// TIA Portal project "一个开关控制两个灯" (V16)

(* hardware
DEVICE "S7-1200 station_1"  S7-1200 Station
   slot 0: "Rack_0"  S7-1200 Rack  Rack  V1.0
   slot 1: "PLC_1"  CPU 1214C DC/DC/DC  6ES7 214-1AG40-0XB0  V4.4
DEVICE "HMI_1"  KTP700 Basic PN
   slot 0: "HMI_1"  KTP700 Basic PN  6AV2 123-2GB03-0AX0  16.0.0.0
   slot 1: "HMI_RT_1"  KTP700 Basic PN  6AV2 123-2GB03-0AX0  16.0.0.0
   slot 5: "HMI_1.IE_CP_1"  PROFINET Interface  16.0.0.0
      slot 1: "PROFINET Interface_1"  PROFINET Interface
         slot 1: "Port_1"  Port
*)

// ===== PLC "PLC_1"  CPU 1214C DC/DC/DC =====

VAR_GLOBAL   // PLC tag table "默认变量表"
   "Tag_1" AT %M0.0 : Bool;
   "Tag_2" AT %M0.1 : Bool;
   "Tag_3" AT %M0.2 : Bool;
   "Tag_4" AT %Q0.1 : Bool;
   "Tag_5" AT %Q0.2 : Bool;
   "Tag_6" AT %M10.0 : Bool;
   "Tag_7" AT %M10.1 : Bool;
   "Tag_8" AT %Q0.7 : Bool;
   "Tag_9" AT %M1.0 : Bool;
   "Tag_10" AT %M1.1 : Bool;
   "Tag_11" AT %M1.2 : Bool;
   "Tag_12" AT %M1.3 : Bool;
   "Tag_13" AT %M1.4 : Bool;
   "Tag_14" AT %Q0.0 : Bool;
   "Tag_15" AT %M2.0 : Bool;
   "Tag_16" AT %M2.1 : Bool;
   "Tag_17" AT %M2.2 : Bool;
   "Tag_18" AT %I0.0 : Bool;
   "Tag_19" AT %Q1.0 : Bool;
   "Tag_20" AT %Q1.1 : Bool;
   "Tag_21" AT %M1.5 : Bool;
   "Tag_22" AT %M1.6 : Bool;
   "Tag_23" AT %M1.7 : Bool;
END_VAR

DATA_BLOCK "数据块_1"   // DB2
{ S7_Optimized_Access := 'TRUE' }
VERSION : 0.1
   VAR
      中间变量1 : Bool;
      中间变量2 : Bool;
      中间变量3 : Bool;
      中间变量4 : Bool;
      中间变量5 : Bool;
      中间变量6 : Bool;
      中间变量7 : Bool;
      中间变量8 : Bool;
      数值 : UDInt := 2;
      上升 : Array[1..10] of Bool;
      下降 : Array[1..10] of Bool;
      中间1 : Array[1..10] of Bool;
   END_VAR
BEGIN
END_DATA_BLOCK

// folder: System blocks/Program resources

DATA_BLOCK "IEC_Counter_0_DB"   // DB1
{ S7_Optimized_Access := 'TRUE' }
AUTHOR : Simatic
FAMILY : IEC
NAME : CNTR
VERSION : 1.0
// stored: InstanceOfName IEC_COUNTER
"IEC_COUNTER"
BEGIN
END_DATA_BLOCK

DATA_BLOCK "IEC_Counter_0_DB_1"   // DB3
{ S7_Optimized_Access := 'TRUE' }
AUTHOR : Simatic
FAMILY : IEC
NAME : CNTR
VERSION : 1.0
// stored: InstanceOfName IEC_COUNTER
"IEC_COUNTER"
BEGIN
END_DATA_BLOCK

DATA_BLOCK "IEC_Counter_0_DB_2"   // DB4
{ S7_Optimized_Access := 'TRUE' }
AUTHOR : Simatic
FAMILY : IEC
NAME : CNTR
VERSION : 1.0
// stored: InstanceOfName IEC_COUNTER
"IEC_COUNTER"
BEGIN
END_DATA_BLOCK

// folder: (top level)

FUNCTION "MHJ-PLC-Lab-Function-S71200" : Void   // FC9000, SCL
{ S7_Optimized_Access := 'TRUE' }
VERSION : 0.1
   VAR_TEMP
      rdTimeReturn : Int;
      outputTime : DTL;
      SyncVal : Byte;
      forVal : Int;
      forVal_2 : Int;
      Value : Byte;
   END_VAR
   VAR CONSTANT
      CompVal : Byte := 16#34;
      Value_01 : Byte := 16#11;
      Value_01_DW : DWord := 16#A165_D992;
      Value_02_DW : DWord := 16#58BE_4401;
   END_VAR
BEGIN

   #Value:=PEEK(area := 16#82,
        dbNumber := 0,
        byteOffset := 511);
   #Value := #Value + 1;

   POKE(area := 16#82,
        dbNumber := 0,
        byteOffset := 511,
        value := #Value);

   POKE(area:=16#81,
        dbNumber:=0,
        byteOffset:=1016,
        value:=#Value_01_DW);
   POKE(area := 16#81,
        dbNumber := 0,
        byteOffset := 1020,
        value := #Value_02_DW);

   POKE(area := 16#81,
        dbNumber := 0,
        byteOffset := 511,
        value := B#16#00);

   FOR #forVal := 0 TO 120 DO
       FOR #forVal_2:=0 TO 10 DO
           #rdTimeReturn:=RD_SYS_T(#outputTime);
           #rdTimeReturn := WR_SYS_T(#outputTime);
           #rdTimeReturn := RD_SYS_T(#outputTime);
           #rdTimeReturn := WR_SYS_T(#outputTime);
       END_FOR;
       #SyncVal:= PEEK(area := 16#81,
                      dbNumber := 0,
                      byteOffset := 511);
       IF #SyncVal = #CompVal THEN
          GOTO M_1;
       END_IF;
   END_FOR;
   RETURN;

   M_1:
   POKE(area := 16#81,
        dbNumber := 0,
        byteOffset := 511,
        value := B#16#0);
END_FUNCTION

ORGANIZATION_BLOCK "Main"   // OB1, LAD, ProgramCycle
TITLE = "Main Program Sweep (Cycle)"
{ S7_Optimized_Access := 'TRUE' }
VERSION : 0.1
   VAR_INPUT
      Initial_Call : Bool;   // Initial call of this OB
      Remanence : Bool;   // =True, if remanent data are available
   END_VAR
   VAR_TEMP   // added for the SCL form of the ladder/FBD networks
      _w1 : Bool;
      _w2 : Bool;
      _w3 : Bool;
      _w4 : Bool;
   END_VAR
BEGIN

REGION Network 1
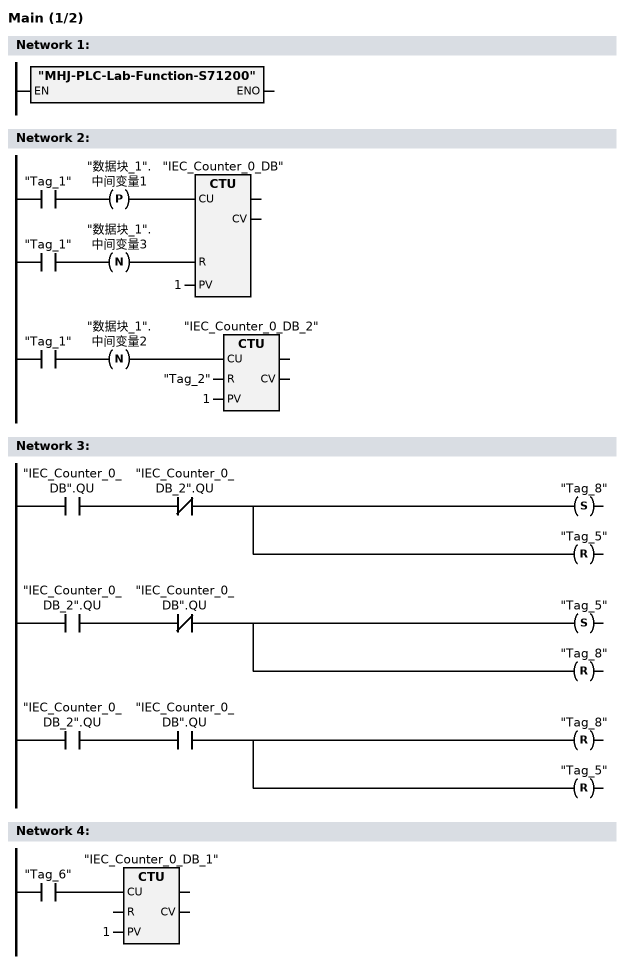
   RUNG wire#powerrail
      "MHJ-PLC-Lab-Function-S71200"()
   END_RUNG
   // the same network as SCL:
   "MHJ-PLC-Lab-Function-S71200"();
END_REGION

REGION Network 2
   #_w1 := "Tag_1" AND NOT "数据块_1".中间变量1;   // rising edge
   "数据块_1".中间变量1 := "Tag_1";
   #_w2 := NOT "Tag_1" AND "数据块_1".中间变量3;   // falling edge
   "数据块_1".中间变量3 := "Tag_1";
   "IEC_Counter_0_DB".CTU(CU := #_w1, R := #_w2, PV := 1);
   #_w3 := NOT "Tag_1" AND "数据块_1".中间变量2;   // falling edge
   "数据块_1".中间变量2 := "Tag_1";
   "IEC_Counter_0_DB_2".CTU(CU := #_w3, R := "Tag_2", PV := 1);
END_REGION

REGION Network 3
   RUNG wire#powerrail
      Contact( "IEC_Counter_0_DB".QU )
      I_Contact( "IEC_Counter_0_DB_2".QU )
      wire#w1
      S_Coil( "Tag_8" )
   END_RUNG
   RUNG wire#w1
      R_Coil( "Tag_5" )
   END_RUNG
   RUNG wire#powerrail
      Contact( "IEC_Counter_0_DB_2".QU )
      I_Contact( "IEC_Counter_0_DB".QU )
      wire#w2
      S_Coil( "Tag_5" )
   END_RUNG
   RUNG wire#w2
      R_Coil( "Tag_8" )
   END_RUNG
   RUNG wire#powerrail
      Contact( "IEC_Counter_0_DB_2".QU )
      Contact( "IEC_Counter_0_DB".QU )
      wire#w3
      R_Coil( "Tag_8" )
   END_RUNG
   RUNG wire#w3
      R_Coil( "Tag_5" )
   END_RUNG
   // the same network as SCL:
   IF "IEC_Counter_0_DB".QU AND NOT "IEC_Counter_0_DB_2".QU THEN
       "Tag_8" := TRUE;
       "Tag_5" := FALSE;
   END_IF;
   IF "IEC_Counter_0_DB_2".QU AND NOT "IEC_Counter_0_DB".QU THEN
       "Tag_5" := TRUE;
       "Tag_8" := FALSE;
   END_IF;
   IF "IEC_Counter_0_DB_2".QU AND "IEC_Counter_0_DB".QU THEN
       "Tag_8" := FALSE;
       "Tag_5" := FALSE;
   END_IF;
END_REGION

REGION Network 4
   "IEC_Counter_0_DB_1".CTU(CU := "Tag_6", PV := 1);
END_REGION

REGION Network 5
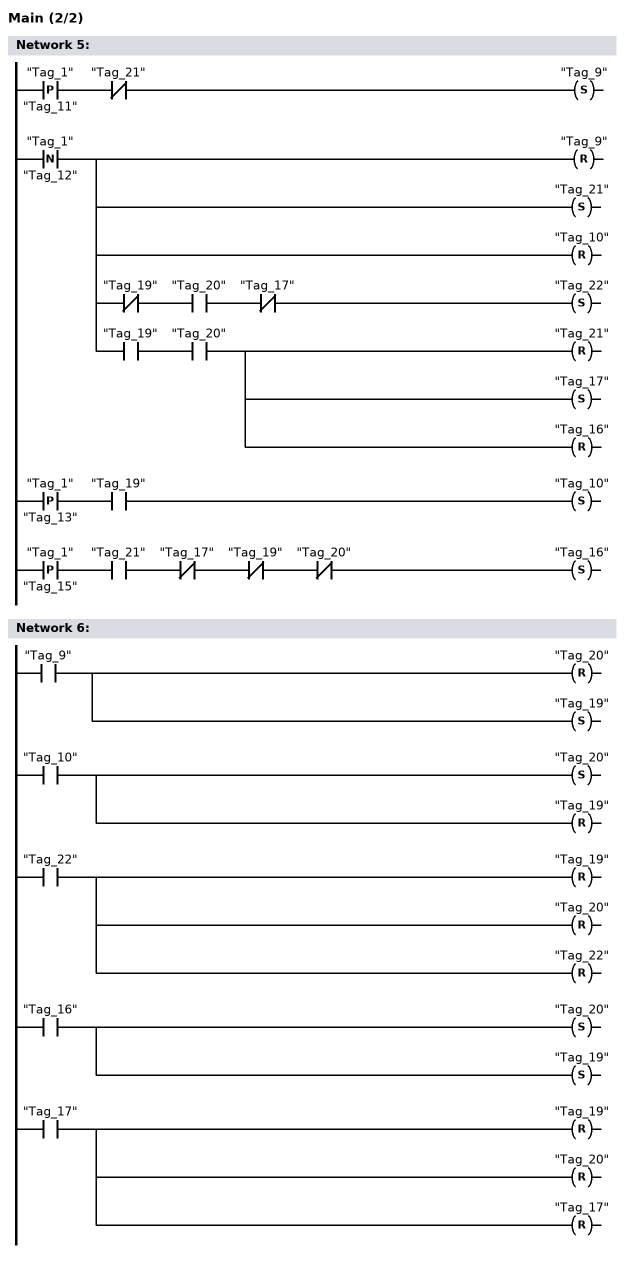
   RUNG wire#powerrail
      P_Contact(operand := "Tag_1", bit := "Tag_11")
      I_Contact( "Tag_21" )
      S_Coil( "Tag_9" )
   END_RUNG
   RUNG wire#powerrail
      N_Contact(operand := "Tag_1", bit := "Tag_12")
      wire#w1
      R_Coil( "Tag_9" )
   END_RUNG
   RUNG wire#w1
      S_Coil( "Tag_21" )
   END_RUNG
   RUNG wire#w1
      R_Coil( "Tag_10" )
   END_RUNG
   RUNG wire#w1
      I_Contact( "Tag_19" )
      Contact( "Tag_20" )
      I_Contact( "Tag_17" )
      S_Coil( "Tag_22" )
   END_RUNG
   RUNG wire#w1
      Contact( "Tag_19" )
      Contact( "Tag_20" )
      wire#w2
      R_Coil( "Tag_21" )
   END_RUNG
   RUNG wire#w2
      S_Coil( "Tag_17" )
   END_RUNG
   RUNG wire#w2
      R_Coil( "Tag_16" )
   END_RUNG
   RUNG wire#powerrail
      P_Contact(operand := "Tag_1", bit := "Tag_13")
      Contact( "Tag_19" )
      S_Coil( "Tag_10" )
   END_RUNG
   RUNG wire#powerrail
      P_Contact(operand := "Tag_1", bit := "Tag_15")
      Contact( "Tag_21" )
      I_Contact( "Tag_17" )
      I_Contact( "Tag_19" )
      I_Contact( "Tag_20" )
      S_Coil( "Tag_16" )
   END_RUNG
   // the same network as SCL:
   #_w1 := "Tag_1" AND NOT "Tag_11";   // rising edge of "Tag_1"
   "Tag_11" := "Tag_1";
   IF #_w1 AND NOT "Tag_21" THEN "Tag_9" := TRUE; END_IF;
   #_w2 := NOT "Tag_1" AND "Tag_12";   // falling edge of "Tag_1"
   "Tag_12" := "Tag_1";
   IF #_w2 THEN
       "Tag_9" := FALSE;
       "Tag_21" := TRUE;
       "Tag_10" := FALSE;
   END_IF;
   IF #_w2 AND NOT "Tag_19" AND "Tag_20" AND NOT "Tag_17" THEN "Tag_22" := TRUE; END_IF;
   IF #_w2 AND "Tag_19" AND "Tag_20" THEN
       "Tag_21" := FALSE;
       "Tag_17" := TRUE;
       "Tag_16" := FALSE;
   END_IF;
   #_w3 := "Tag_1" AND NOT "Tag_13";   // rising edge of "Tag_1"
   "Tag_13" := "Tag_1";
   IF #_w3 AND "Tag_19" THEN "Tag_10" := TRUE; END_IF;
   #_w4 := "Tag_1" AND NOT "Tag_15";   // rising edge of "Tag_1"
   "Tag_15" := "Tag_1";
   IF #_w4 AND "Tag_21" AND NOT "Tag_17" AND NOT "Tag_19" AND NOT "Tag_20" THEN "Tag_16" := TRUE; END_IF;
END_REGION

REGION Network 6
   RUNG wire#powerrail
      Contact( "Tag_9" )
      wire#w1
      R_Coil( "Tag_20" )
   END_RUNG
   RUNG wire#w1
      S_Coil( "Tag_19" )
   END_RUNG
   RUNG wire#powerrail
      Contact( "Tag_10" )
      wire#w2
      S_Coil( "Tag_20" )
   END_RUNG
   RUNG wire#w2
      R_Coil( "Tag_19" )
   END_RUNG
   RUNG wire#powerrail
      Contact( "Tag_22" )
      wire#w3
      R_Coil( "Tag_19" )
   END_RUNG
   RUNG wire#w3
      R_Coil( "Tag_20" )
   END_RUNG
   RUNG wire#w3
      R_Coil( "Tag_22" )
   END_RUNG
   RUNG wire#powerrail
      Contact( "Tag_16" )
      wire#w4
      S_Coil( "Tag_20" )
   END_RUNG
   RUNG wire#w4
      S_Coil( "Tag_19" )
   END_RUNG
   RUNG wire#powerrail
      Contact( "Tag_17" )
      wire#w5
      R_Coil( "Tag_19" )
   END_RUNG
   RUNG wire#w5
      R_Coil( "Tag_20" )
   END_RUNG
   RUNG wire#w5
      R_Coil( "Tag_17" )
   END_RUNG
   // the same network as SCL:
   IF "Tag_9" THEN
       "Tag_20" := FALSE;
       "Tag_19" := TRUE;
   END_IF;
   IF "Tag_10" THEN
       "Tag_20" := TRUE;
       "Tag_19" := FALSE;
   END_IF;
   IF "Tag_22" THEN
       "Tag_19" := FALSE;
       "Tag_20" := FALSE;
       "Tag_22" := FALSE;
   END_IF;
   IF "Tag_16" THEN
       "Tag_20" := TRUE;
       "Tag_19" := TRUE;
   END_IF;
   IF "Tag_17" THEN
       "Tag_19" := FALSE;
       "Tag_20" := FALSE;
       "Tag_17" := FALSE;
   END_IF;
END_REGION
END_ORGANIZATION_BLOCK

(* ===== HMI "HMI_RT_1" =====
system functions are stored by id; their names below are inferred from use
connection "HMI_连接_1": ETHERNET, SMART_S7_1200_OMS

HMI tags "默认变量表"
   "Tag_ScreenNumber" : UInt, internal
   "Tag_5" : Bool = PLC Tag_5 AT %Q0.2, 1 s
   "Tag_8" : Bool = PLC Tag_8 AT %Q0.7, 1 s
   "Tag_1" : Bool = PLC Tag_1 AT %M0.0, 1 s
   "Tag_4" : Bool = PLC Tag_4 AT %Q0.1, 1 s
   "Tag_19" : Bool = PLC Tag_19 AT %Q1.0, 1 s
   "Tag_20" : Bool = PLC Tag_20 AT %Q1.1, 1 s

Template "模板_1" 800x480
   Button "退出" at 714,429 size 71x50; TextOff '退出'; PictureOff "ExitRuntime_KTP700_Basic_PN_TR"; PictureOn "ExitRuntime_KTP700_Basic_PN_TR"
      on Release: StopRuntime(0)
   Button "Template_Button" at 614,429 size 71x50; TextOff 'Text'
   Button "Template_Button_1" at 514,429 size 71x50; TextOff 'Text'
   Button "Template_Button_2" at 414,429 size 71x50; TextOff 'Text'
   Button "Template_Button_3" at 314,429 size 71x50; TextOff 'Text'
   Button "Template_Button_4" at 214,429 size 71x50; TextOff 'Text'
   Button "Template_Button_5" at 114,429 size 71x50; TextOff 'Text'
   Button "起始画面" at 14,429 size 71x50; TextOff '起始画面'; PictureOff "NavigateHome_KTP700_Basic_PN_TR"; PictureOn "NavigateHome_KTP700_Basic_PN_TR"
      on Release: ActivateScreen("根画面", 0)
   SymbolicIOField "Symbolic_IO_Field_Screen" at 93,9 size 600x33; TextOff '0'; TextOn '1'; TextList "TextList_ScreenNames"
      ProcessValue <- "Tag_ScreenNumber"
      on Change: ActivateScreenByNumber("Tag_ScreenNumber", 0)
   DateTimeField "HmiScreenItemData" at 695,25 size 105x25
   DateTimeField "HmiScreenItemData_1" at 695,0 size 105x25
   GraphicView "Logo" at 0,0 size 91x51; Picture "HMI_1 的 Logo"

screen "根画面" 800x480, template "模板_1"
   on GenerateScreen: SetTag("Tag_ScreenNumber", 1)
   Button "按钮_1" at 192,250 size 96x32; TextOff '开关'
      on Click: InvertBit("Tag_1")
   Circle "圆_1" at 454,97 size 48x48
      Appearance <- "Tag_19"
   Circle "圆_2" at 454,176 size 48x48
      Appearance <- "Tag_20"
*)